// TwinCAT 3 PLC project Plc
// Title: Template.Essentials
// Company: Template.Essentials
// ProjectVersion: 0.0.0.1
// ProgramVersion: 3.1.4023.0
// libraries:
//   Tc2_Standard, * (Beckhoff Automation GmbH)
//   Tc2_System, * (Beckhoff Automation GmbH)
//   Tc3_Module, * (Beckhoff Automation GmbH)
// project tree:
//   DUTs/ stBools.TcDUT, stEntity.TcDUT, stSettings.TcDUT, stTreeStruct.TcDUT
//   / PlcTask.TcTTO
//   POUs/CSharp/ CSharpMethod.TcPOU
//   POUs/Data/ DataManager.TcPOU
//   POUs/Email/ fbEmail.TcPOU
//   POUs/ MAIN.TcPOU, stPrograms.TcDUT
//   POUs/REST/ fbRest.TcPOU
//   POUs/SMS/ fbSms.TcPOU
//   POUs/Sorter/ RemoteSorting.TcPOU
// real-time tasks:
//   TASK PlcTask: cycle T#10ms, priority 20, ADS port 350

CONFIGURATION Plc
    RESOURCE PLC ON TwinCAT3
        TASK PlcTask(INTERVAL := T#10ms, PRIORITY := 20);
        PROGRAM MAIN WITH PlcTask : MAIN;
    END_RESOURCE
END_CONFIGURATION

// ---- DUTs/stBools.TcDUT
{attribute wpf [Container(Layout.Stack)]}
TYPE stBools :
STRUCT
	BoolOne :BOOL;
	BoolTwo:BOOL;
	BoolThree:BOOL;
	BoolFive:BOOL;
END_STRUCT
END_TYPE

// ---- DUTs/stEntity.TcDUT
TYPE stEntity :
STRUCT
	
END_STRUCT
END_TYPE

// ---- DUTs/stSettings.TcDUT
TYPE stSettings EXTENDS stEntity :
STRUCT
	One:BOOL;
	Two:BOOL;
	Another:STRING;
	ThisOne:STRING;
	bools :stBools;
	trees : stTreeStruct;
	xbools :stBools;
	atrees : stTreeStruct;
	sbools :stBools;
	ttrees : stTreeStruct;
END_STRUCT
END_TYPE

// ---- DUTs/stTreeStruct.TcDUT
{attribute wpf [Container(Layout.Stack)]}
TYPE stTreeStruct :
STRUCT
	One:BOOL;
	Two:BOOL;
	Another:STRING;
	ThisOne:STRING;
	ANumberWouldBeCool:INT;
	Bools : stBools;
END_STRUCT
END_TYPE

// ---- POUs/stPrograms.TcDUT
	{attribute wpf [Container(Layout.Tabs)]}
TYPE stPrograms :
STRUCT	 
	{attribute wpf [Container(Layout.Stack)]}
	EmailSender : fbEmail;
	{attribute wpf [Container(Layout.Stack)]}
	Sorting : RemoteSorting;
	{attribute wpf [Container(Layout.Stack)]}
	Data : DataManager;
	{attribute wpf [Container(Layout.Stack)]}
	TextMsg : fbSms;
	{attribute wpf [Container(Layout.Stack)]}
	RestCall :fbRest;
END_STRUCT
END_TYPE

// ---- POUs/MAIN.TcPOU
PROGRAM MAIN
VAR
	{attribute wpf [Container(Layout.Tabs)]}
	App :stPrograms;
END_VAR

App.EmailSender();
App.Sorting();
App.Data();
App.TextMsg();
App.RestCall();

END_PROGRAM

// ---- POUs/CSharp/CSharpMethod.TcPOU
FUNCTION_BLOCK CSharpMethod
VAR
	InvokeRequested : BOOL;
	InvokeInProgress : BOOL;
	InvokeDone : BOOL;
	InvokeError : BOOL;
	ErrorMessage :STRING;
	CommandId : STRING;
END_VAR

METHOD Invoke : BOOL
IF  NOT InvokeRequested AND 
	NOT InvokeInProgress 
THEN 
	InvokeRequested := TRUE; // Inxton listens to this change
	InvokeDone :=FALSE;
	InvokeError :=FALSE; 
END_IF

// Inxton will set the execution to InProgress.
IF InvokeInProgress THEN
	//Inxton will set the Done after the execution finished. 	
	IF InvokeDone THEN
		InvokeInProgress := FALSE;
		InvokeRequested := FALSE;
		Invoke := TRUE;
		RETURN;
	END_IF
	
END_IF
END_METHOD

END_FUNCTION_BLOCK

// ---- POUs/Data/DataManager.TcPOU
FUNCTION_BLOCK DataManager
VAR
	Settings : stSettings;
	{attribute addProperty Name "Save to database" }
	SaveSettings : CSharpMethod;
	{attribute clr [RenderIgnore()]}
	Invoke :BOOL;
END_VAR

IF Invoke THEN
	IF Save() THEN
		Invoke :=FALSE;	
	END_IF
END_IF

METHOD Save : BOOL
VAR_INPUT
END_VAR
Save := SaveSettings.Invoke();
END_METHOD

END_FUNCTION_BLOCK

// ---- POUs/Email/fbEmail.TcPOU
FUNCTION_BLOCK fbEmail
VAR
	Recipient:STRING := 'jozef.chmelar@inxton.com';
	Subject:STRING := 'Hello PLC Subject';
	Content : STRING := 'This email is from the PLC!';
	{attribute addProperty Name "Send email" }
	SendEmail : CSharpMethod;
	{attribute clr [RenderIgnore()]}
	StartSending : BOOL;
END_VAR

IF StartSending THEN
	IF SendEmail.Invoke() THEN
		StartSending :=FALSE;	
	END_IF
END_IF

END_FUNCTION_BLOCK

// ---- POUs/REST/fbRest.TcPOU
FUNCTION_BLOCK fbRest
VAR
	ToAnalyse : STRING := 'I think you$'re a great person! I think he$'s much worse than you are.';
	AnalysisResult:STRING;
	{attribute addProperty Name "Analyse sentiment" }
	RestCall : CSharpMethod;
	{attribute clr [RenderIgnore()]}
	StartSending : BOOL;
END_VAR

IF StartSending THEN
	IF RestCall.Invoke() THEN
		StartSending :=FALSE;	
	END_IF
END_IF

END_FUNCTION_BLOCK

// ---- POUs/SMS/fbSms.TcPOU
FUNCTION_BLOCK fbSms
VAR
	Recipient:STRING := '+15558675310';
	Content : STRING := ' This a test message is from the PLC!';
	{attribute addProperty Name "Send text message" }
	SendTextMessage : CSharpMethod;
	{attribute clr [RenderIgnore()]}
	StartSending : BOOL;
END_VAR

IF StartSending THEN
	IF SendTextMessage.Invoke() THEN
		StartSending :=FALSE;	
	END_IF
END_IF

END_FUNCTION_BLOCK

// ---- POUs/Sorter/RemoteSorting.TcPOU
FUNCTION_BLOCK RemoteSorting
VAR
	MyArray : ARRAY [0..10] OF INT;
	MyArrayToString : STRING;
	{attribute addProperty Name "Sort" }
	Sort : CSharpMethod;
	InitArray : BOOL := TRUE;
	{attribute clr [RenderIgnore()]}	
	i:INT;
END_VAR

IF InitArray THEN
	FOR i := 0 TO 10  DO
		MyArray[i] :=  10-i;
	END_FOR;
	InitArray :=FALSE;
END_IF

MyArrayToString := '';
FOR i := 0 TO 10  DO
	MyArrayToString := CONCAT(MyArrayToString, INT_TO_STRING(MyArray[i]) );
	MyArrayToString := CONCAT(MyArrayToString,', ');
END_FOR;

END_FUNCTION_BLOCK
